	16#818E:           
		F_TcError:= 'Master/Slave sync position incompatible with sync direction The given sync positions require the slave moving in a direction which is not allowed while in synchronization phase';
                       
	16#8191:           
		F_TcError:= 'Unexpected axis state At least one axis has an unexpected state This may occur if a group reset is active and an axis error occurs after the respective axis was successfully reset';
                       
	16#8192:           
		F_TcError:= 'Invalid reference system The reference system is unknown or invalid for this application';
                       
	16#8193:           
		F_TcError:= 'Position not in reference system The position is outside of the specified reference system';
                       
	16#8194:           
		F_TcError:= 'A previous command is blocking execution A previous command is still ongoing and simultaneous execution of both commands is impossible';
                       
	16#8198:           
		F_TcError:= 'Invalid index The used index does not exist or is invalid';
                       
	16#8199:           
		F_TcError:= 'Command not allowed The command is not allowed in the current configuration';
                       
	16#8F2F:           
		F_TcError:= 'Internal Error';
                       
	16#8F50:           
		F_TcError:= 'Internal Error';
                       
	16#8f56:           
		F_TcError:= 'Internal Error';
                       
	16#8F59:           
		F_TcError:= 'Internal Error';
                       
	16#8F5C:           
		F_TcError:= 'Internal Error';
                       
	16#8F62:           
		F_TcError:= 'Internal Error';
                       
	16#8F65:           
		F_TcError:= 'Internal Error';
                       
	16#8F68:           
		F_TcError:= 'Internal Error';
                       
	16#8FCE:           
		F_TcError:= 'Internal Error';
                       
	16#8FD0:           
		F_TcError:= 'Internal Error';
                       
	16#8FFFF:           
		F_TcError:= 'Internal Error';

{endregion}	
END_CASE

END_FUNCTION
